// TIA Portal V21 export
DATA_BLOCK "Sequenza"   // DB22
{ S7_Optimized_Access := 'TRUE' }
// stored: MemoryReserve 100
   VAR RETAIN
      S : Array[0.."K_NumSequenza"] of "Std_Sequenza";
   END_VAR
   VAR
      Hmi : Struct
         PassoAttuale : Int := 3;
         SequenzaAttuale : Int := 2;
      END_STRUCT;
   END_VAR
BEGIN
   // S[0] : Non usare
   S[0].Prm.Passo[0..25].Durata.IN := FALSE;
   S[0].Prm.Passo[0..25].Durata.O := FALSE;
   S[0].Prm.Passo[0..25].Durata.Preset := 0.0;
   S[0].Prm.Passo[0..25].Durata.TempoTrascorso := 0.0;
   S[0].Hmi.Stato := 0;
   S[0].Hmi.BloccaAvanzamento := FALSE;
   S[0].Hmi.ArrestaSequenza := FALSE;
   S[0].Hmi.AvviaSequenza := FALSE;
   S[0].Hmi.AvviaSequenzaDisabilitato := FALSE;
   S[0].Hmi.TempoRimanente := 0.0;
   S[0].Hmi.SaltaPasso.Abilitato := FALSE;
   S[0].Hmi.SaltaPasso.Richiesto := FALSE;
   S[0].Hmi.AttendiAckOpertore.AbilitaFunz := FALSE;
   S[0].Hmi.AttendiAckOpertore.AckOperatore := FALSE;
   S[0].Hmi.Diagnostica.AttesaValvola := 0;
   S[0].Hmi.Diagnostica.AttesaMotore := 0;
   S[0].Hmi.Diagnostica.AttesaAnalogica := 0;
   S[0].Hmi.Diagnostica.AttesaPortata := 0;
   S[0].Hmi.Diagnostica.AttesaExtCondi := FALSE;
   S[0].Hmi.Diagnostica.AttesaTempo := FALSE;
   S[0].Hmi.Diagnostica.PassoNonAbilitato := FALSE;
   S[0].Dati.PassoAttuale := 0;
   S[0].Dati.TutteLeUtenzeInPosizione := FALSE;
   S[0].Dati.AbilitazionePasso := FALSE;
   S[0].Dati.TempoRimanente := 0.0;
   S[0].Dati.TempoTerminato_AttesaCondExt := FALSE;
   S[0].Dati.ResettaTuttiFlipFlop := FALSE;
   S[0].Dati.MemoPassoAttuale := 0;
   S[0].Dati.PrimoGiroPasso := FALSE;
   S[0].Allarmi."A"[0].Abilitato := FALSE;
   S[0].Allarmi."A"[0].Stato := FALSE;
   S[0].Allarmi."A"[0].Silenziato := FALSE;
   S[0].Allarmi."A"[0].EnWarnHmi := FALSE;
   S[0].Allarmi."A"[0].EnCadutaCiclo := FALSE;
   S[0].Allarmi.WordHMI := 16#0000;
   S[0].Out.SequenzaAvviata := FALSE;
   S[0].Out.Passo[0..25].Attivo := FALSE;
END_DATA_BLOCK
